(* CoDeSys 2.3 export: MB_GLOBALVAR.EXP *)

(* Global variable list: MB_GlobalVar *)
VAR_GLOBAL
	(*Modbusmaster*)
	ModbusMaster: ModbusRtuMaster_KL6x22B; (*Declaratie is globaal omdat deze bouwsteen door meerdere functieblokken wordt gebruikt*)
	gv_iMasterInGebruikDoor:INT;
END_VAR
